// TIA Portal V19 export
DATA_BLOCK "HMI Tags"   // DB72
{ S7_Optimized_Access := 'TRUE' }
// stored: MemoryReserve 100
   VAR
      ControlAutoSelect : Bool := FALSE;
      ControlAutoStart : Bool := FALSE;
      ControlAutoStop : Bool := FALSE;
      AutoRunning : Bool := FALSE;
      ResetAlarms : Bool := FALSE;
   END_VAR
   VAR RETAIN
      "Select Input" : Struct
         "Input 1" : Int := 1;
         "Input 2" : Int := 10;
         "Input 3" : Int := 0;
         "Input 4" : Int := 0;
         "Input 5" : Int := 0;
         "Input 6" : Int := 0;
         "Input 7" : Int := 0;
         "Input 8" : Int := 0;
         "Input 9" : Int := 0;
         "Input 10" : Int := 0;
         "Input 11" : Int := 0;
         "Input 12" : Int := 0;
         "Input 13" : Int := 0;
         "Input 14" : Int := 0;
      END_STRUCT;
      "Selected Input" : Struct
         "Input 1" : Int := 0;
         "Input 2" : Int := 0;
         "Input 3" : Int := 0;
         "Input 4" : Int := 0;
         "Input 5" : Int := 0;
         "Input 6" : Int := 0;
         "Input 7" : Int := 0;
         "Input 8" : Int := 0;
         "Input 9" : Int := 0;
         "Input 10" : Int := 0;
         "Input 11" : Int := 0;
         "Input 12" : Int := 0;
         "Input 13" : Int := 0;
         "Input 14" : Int := 0;
      END_STRUCT;
      "Select Output" : Struct
         "output 1" : Int := 0;
         "output 2" : Int := 0;
         "output 3" : Int := 0;
         "output 4" : Int := 0;
         "output 5" : Int := 0;
         "output 6" : Int := 0;
         "output 7" : Int := 0;
         "output 8" : Int := 0;
         "output 9" : Int := 0;
         "output 10" : Int := 0;
      END_STRUCT;
      "Selected Output" : Struct
         "output 1" : Int := 0;
         "output 2" : Int := 0;
         "output 3" : Int := 0;
         "output 4" : Int := 0;
         "output 5" : Int := 0;
         "output 6" : Int := 0;
         "output 7" : Int := 0;
         "output 8" : Int := 0;
         "output 9" : Int := 0;
         "output 10" : Int := 0;
      END_STRUCT;
      LinePressure : "AnalogScale";
      BufferLevel { S7_SetPoint := 'True'} : "AnalogScale";
      SpareAN1 { S7_SetPoint := 'True'} : "AnalogScale";
      SpareAN2 { S7_SetPoint := 'True'} : "AnalogScale";
      CoolOverRunValue { S7_SetPoint := 'True'} : Time := T#1M;
      Pump_Control : "VFD_Control";
   END_VAR
   VAR
      ResetMotorFault : Bool := FALSE;
   END_VAR
   VAR RETAIN
      LinePressureMin { S7_SetPoint := 'True'} : Real := 0.0;
      LinePressureMax : Real := 0.0;
      LinePressureSP : Real := 0.0;
   END_VAR
   VAR
      "Manual Run Motor" : Bool := FALSE;
   END_VAR
   VAR RETAIN
      ModeOneShot : Bool := FALSE;
      ModeRepeat : Bool := TRUE;
      ModeOneShotTime : Bool := FALSE;
      ModeRepeatTime : Bool := FALSE;
      ModeContinous : Bool := FALSE;
   END_VAR
   VAR
      StartDose : Bool := FALSE;
   END_VAR
   VAR RETAIN
      "Required Dose" : Real := 1000.0;
      InflightVal : Real := 0.0;
      CalcDose : Real := 1000.0;
      DoseTime : Time := T#0MS;
      IntervalTime : Time := T#5S;
      IBC : "Valve";
      Flowmeter { S7_SetPoint := 'True'} : "Valve";
      Dose { S7_SetPoint := 'True'} : "Valve";
      Pump { S7_SetPoint := 'True'} : "Valve";
      WriteLogs { S7_SetPoint := 'True'} : Bool := FALSE;
   END_VAR
   VAR
      alarms : DWord := 16#0000_0000;
   END_VAR
   VAR RETAIN
      MinimumLinePressure : Real := 0.0;
      MaximumLinePressure : Real := 12.0;
      SystemEnables : Struct
         "Flowmeter Fitted" : Bool := TRUE;
         LinePressureFitted : Bool := TRUE;
         FlowmeterTemperatureFitted : Bool := TRUE;
         IBCFitted : Bool := FALSE;
         IBCValveFitted : Bool := FALSE;
         FlowmeterValveFitted : Bool := TRUE;
         "Buffer LevelFitted" : Bool := FALSE;
         PumpValveFitted : Bool := FALSE;
         DoseValveFitted : Bool := TRUE;
         ForcedCoolingFitted : Bool := TRUE;
         BufferValveFitted : Bool := FALSE;
      END_STRUCT;
      TemperatureLowSP : Real := 15.0;
      TemperatureHighSP : Real := 30.0;
      BufferHopperMinLVL : Real := 0.0;
      BufferHopperMaxLVL : Real := 0.0;
      BufferHopperLVLSP : Real := 0.0;
      HMISettingsLock : Bool := FALSE;
   END_VAR
   VAR
      DoseState : Int := 0;
   END_VAR
   VAR RETAIN
      DoseWaiting : Time := T#5S;
   END_VAR
   VAR
      FMActualCount : Real := 0.0;
      DoseActTime : Time := T#0MS;
      FmTemperature : Real := 17.8934;
   END_VAR
BEGIN
   LinePressure.AnalogMin := 0;
   LinePressure.AnalogMax := 27648;
   LinePressure.ScaledMIN := 0.0;
   LinePressure.ScaledMax := 11.0;
   LinePressure.ScaledSensor := 0.06127026;
   BufferLevel.AnalogMin := 0;
   BufferLevel.AnalogMax := 0;
   BufferLevel.ScaledMIN := 0.0;
   BufferLevel.ScaledMax := 0.0;
   BufferLevel.ScaledSensor := 0.0;
   SpareAN1.AnalogMin := 0;
   SpareAN1.AnalogMax := 0;
   SpareAN1.ScaledMIN := 0.0;
   SpareAN1.ScaledMax := 0.0;
   SpareAN1.ScaledSensor := 0.0;
   SpareAN2.AnalogMin := 0;
   SpareAN2.AnalogMax := 0;
   SpareAN2.ScaledMIN := 0.0;
   SpareAN2.ScaledMax := 0.0;
   SpareAN2.ScaledSensor := 0.0;
   Pump_Control.NameplateSpeed := 710.0;
   Pump_Control.AutoSpeedSP := 50.0;
   Pump_Control.DriveIsRunning := FALSE;
   Pump_Control.ActualSpeed := 0.0;
   Pump_Control.AxisActive := FALSE;
   Pump_Control.LockoutActive := FALSE;
   Pump_Control.ErrorPResent := FALSE;
   Pump_Control.HMI_VFD_Fault := 0;
   Pump_Control.HMI_Error_Present := FALSE;
   Pump_Control.VFDFaultCode := 0;
   Pump_Control.MotorState := 0;
   Pump_Control.Actual_Current := 0.0007141113;
   Pump_Control.Actual_torque := 0.0;
   Pump_Control.Peak_Current := 0.0;
   Pump_Control.Peak_torque := 0.0;
   IBC.ManOpen := FALSE;
   IBC.FeebackFitted := FALSE;
   IBC.ValveisOpen := FALSE;
   IBC.ValveisClosed := FALSE;
   IBC.ValveAngle := 0.0;
   IBC.FeedbackFaultTime := T#0MS;
   Flowmeter.ManOpen := FALSE;
   Flowmeter.FeebackFitted := FALSE;
   Flowmeter.ValveisOpen := FALSE;
   Flowmeter.ValveisClosed := TRUE;
   Flowmeter.ValveAngle := 90.0;
   Flowmeter.FeedbackFaultTime := T#0MS;
   Dose.ManOpen := FALSE;
   Dose.FeebackFitted := FALSE;
   Dose.ValveisOpen := FALSE;
   Dose.ValveisClosed := TRUE;
   Dose.ValveAngle := 90.0;
   Dose.FeedbackFaultTime := T#0MS;
   Pump.ManOpen := FALSE;
   Pump.FeebackFitted := FALSE;
   Pump.ValveisOpen := FALSE;
   Pump.ValveisClosed := FALSE;
   Pump.ValveAngle := 0.0;
   Pump.FeedbackFaultTime := T#0MS;
END_DATA_BLOCK
